(* Logix 5000 project; controller R1USB70001_CWRU_Scenario_Gen_20111116 vendor 1 type 14 code 54 rev 19.11; software revision 19.01; part 2 of 6 *)
(* tags used below, declared in another part *)
   ControlModePv : ControlModePv;
   DiscreteOutputsPv : DiscreteOutputsPv;
   ExecutePv : ExecutePv;
   Alternate_Control_Buffer : Output_Array;   // Array of bit-defined words from Alternate (external) Control source
   AP_GP_CH_SG1 : ALIAS FOR ACNR_GP_SG_N2:1:O.2;
   AP_GP_CH_SG2 : ALIAS FOR ACNR_GP_SG_N2:1:O.3;
   AP_GP_SR_SG1 : ALIAS FOR ACNR_GP_SG_N2:1:O.0;
   AP_GP_SR_SG2 : ALIAS FOR ACNR_GP_SG_N2:1:O.1;
   AS_SP_L1_SG1 : ALIAS FOR ACNR_SP_SG_N3:1:O.0;
   AS_SP_L1_SG2 : ALIAS FOR ACNR_SP_SG_N3:1:O.1;
   AS_SP_L2_SG1 : ALIAS FOR ACNR_SP_SG_N3:1:O.2;
   AS_SP_L2_SG2 : ALIAS FOR ACNR_SP_SG_N3:1:O.3;
   BuildTableIndex : DINT;
   CalcRemainTimeIndex : DINT;
   CalcTotalTimeIndex : DINT;
   CL_GP_SC_SG1 : ALIAS FOR ACNR_GP_SG_N2:5:O.0;
   CL_GP_SC_SG2 : ALIAS FOR ACNR_GP_SG_N2:5:O.1;
   CL_GP_SF_SG1 : ALIAS FOR ACNR_GP_SG_N2:5:O.2;
   CL_GP_SF_SG2 : ALIAS FOR ACNR_GP_SG_N2:5:O.3;
   CL_GP_WF_SG1 : ALIAS FOR ACNR_GP_SG_N2:5:O.6;
   CL_GP_WF_SG2 : ALIAS FOR ACNR_GP_SG_N2:5:O.7;
   CL_GP_WT_SG1 : ALIAS FOR ACNR_GP_SG_N2:5:O.4;
   CL_GP_WT_SG2 : ALIAS FOR ACNR_GP_SG_N2:5:O.5;
   ControlMode : ControlModePub;
   Execute : ExecutePub;
   HMI : HMIPub;
   IL_GP_SC_SG1 : ALIAS FOR ACNR_GP_SG_N2:6:O.0;
   IL_GP_SC_SG2 : ALIAS FOR ACNR_GP_SG_N2:6:O.1;
   IL_GP_SF_SG1 : ALIAS FOR ACNR_GP_SG_N2:6:O.2;
   IL_GP_SF_SG2 : ALIAS FOR ACNR_GP_SG_N2:6:O.3;
   IL_GP_WF_SG1 : ALIAS FOR ACNR_GP_SG_N2:6:O.6;
   IL_GP_WF_SG2 : ALIAS FOR ACNR_GP_SG_N2:6:O.7;
   IL_GP_WT_SG1 : ALIAS FOR ACNR_GP_SG_N2:6:O.4;
   IL_GP_WT_SG2 : ALIAS FOR ACNR_GP_SG_N2:6:O.5;
   RL_GP_SC_SG1 : ALIAS FOR ACNR_GP_SG_N2:4:O.0;
   RL_GP_SC_SG2 : ALIAS FOR ACNR_GP_SG_N2:4:O.1;
   RL_GP_SF_SG1 : ALIAS FOR ACNR_GP_SG_N2:4:O.2;
   RL_GP_SF_SG2 : ALIAS FOR ACNR_GP_SG_N2:4:O.3;
   RL_GP_WF_SG1 : ALIAS FOR ACNR_GP_SG_N2:4:O.6;
   RL_GP_WF_SG2 : ALIAS FOR ACNR_GP_SG_N2:4:O.7;
   RL_GP_WT_SG1 : ALIAS FOR ACNR_GP_SG_N2:4:O.4;
   RL_GP_WT_SG2 : ALIAS FOR ACNR_GP_SG_N2:4:O.5;
   RL_LP_B1_L1_SG1 : ALIAS FOR ACNR_RP_SG_N4:1:O.2;
   RL_LP_B1_L1_SG2 : ALIAS FOR ACNR_RP_SG_N4:1:O.3;
   RL_LP_B1_L2_SG1 : ALIAS FOR ACNR_RP_SG_N4:1:O.4;
   RL_LP_B1_L2_SG2 : ALIAS FOR ACNR_RP_SG_N4:1:O.5;
   RL_LP_B1_L3_SG1 : ALIAS FOR ACNR_RP_SG_N4:1:O.6;
   RL_LP_B1_L3_SG2 : ALIAS FOR ACNR_RP_SG_N4:1:O.7;
   RL_LP_B1_L4_SG1 : ALIAS FOR ACNR_RP_SG_N4:2:O.0;
   RL_LP_B1_L4_SG2 : ALIAS FOR ACNR_RP_SG_N4:2:O.1;
   RL_LP_B1_L5_SG1 : ALIAS FOR ACNR_RP_SG_N4:2:O.2;
   RL_LP_B1_SG : ALIAS FOR ACNR_RP_SG_N4:1:O.1;
   RL_LP_ML_SG : ALIAS FOR ACNR_RP_SG_N4:1:O.0;
   SC_GP_BT_SG1 : ALIAS FOR ACNR_GP_SG_N2:3:O.0;
   SC_GP_BT_SG2 : ALIAS FOR ACNR_GP_SG_N2:3:O.1;
   SC_GP_GD_SG1 : ALIAS FOR ACNR_GP_SG_N2:3:O.2;
   SC_GP_GD_SG2 : ALIAS FOR ACNR_GP_SG_N2:3:O.3;
   SC_SP_LN_SG1 : ALIAS FOR ACNR_SP_SG_N3:2:O.2;
   SC_SP_LN_SG2 : ALIAS FOR ACNR_SP_SG_N3:2:O.3;
   Scenario : Scenario_Def[100];
   SF_GP_BT_SG1 : ALIAS FOR ACNR_GP_SG_N2:2:O.4;
   SF_GP_BT_SG2 : ALIAS FOR ACNR_GP_SG_N2:2:O.5;
   SF_GP_GD_SG1 : ALIAS FOR ACNR_GP_SG_N2:2:O.6;
   SF_GP_GD_SG2 : ALIAS FOR ACNR_GP_SG_N2:2:O.7;
   SF_SP_LN_SG1 : ALIAS FOR ACNR_SP_SG_N3:2:O.0;
   SF_SP_LN_SG2 : ALIAS FOR ACNR_SP_SG_N3:2:O.1;
   TimeTblStepNmbr : DINT;
   WF_GP_BT_SG1 : ALIAS FOR ACNR_GP_SG_N2:1:O.4;
   WF_GP_BT_SG2 : ALIAS FOR ACNR_GP_SG_N2:1:O.5;
   WF_GP_GD_SG1 : ALIAS FOR ACNR_GP_SG_N2:1:O.6;
   WF_GP_GD_SG2 : ALIAS FOR ACNR_GP_SG_N2:1:O.7;
   WF_SP_LN_SG1 : ALIAS FOR ACNR_SP_SG_N3:1:O.4;
   WF_SP_LN_SG2 : ALIAS FOR ACNR_SP_SG_N3:1:O.5;
   WT_GP_BT_SG1 : ALIAS FOR ACNR_GP_SG_N2:2:O.0;
   WT_GP_BT_SG2 : ALIAS FOR ACNR_GP_SG_N2:2:O.1;
   WT_GP_GD_SG1 : ALIAS FOR ACNR_GP_SG_N2:2:O.2;
   WT_GP_GD_SG2 : ALIAS FOR ACNR_GP_SG_N2:2:O.3;
   WT_SP_LN_SG1 : ALIAS FOR ACNR_SP_SG_N3:1:O.6;
   WT_SP_LN_SG2 : ALIAS FOR ACNR_SP_SG_N3:1:O.7;
(* MainProgram, continued *)

ROUTINE BuildTimeTableStep   (* ladder *)
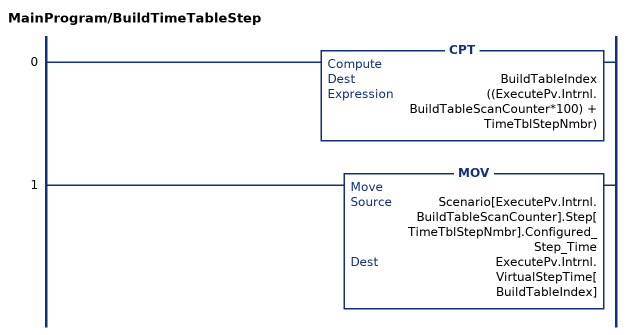
   0: CPT(BuildTableIndex,((ExecutePv.Intrnl.BuildTableScanCounter*100) + TimeTblStepNmbr));
   1: MOV(Scenario[ExecutePv.Intrnl.BuildTableScanCounter].Step[TimeTblStepNmbr].Configured_Step_Time,ExecutePv.Intrnl.VirtualStepTime[BuildTableIndex]);
END_ROUTINE

ROUTINE CalculateCampaignTime   (* ladder *)
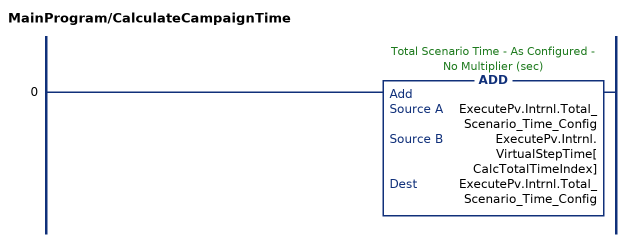
   0: ADD(ExecutePv.Intrnl.Total_Scenario_Time_Config,ExecutePv.Intrnl.VirtualStepTime[CalcTotalTimeIndex],ExecutePv.Intrnl.Total_Scenario_Time_Config);
END_ROUTINE

ROUTINE CalculateRemainingTime   (* ladder *)
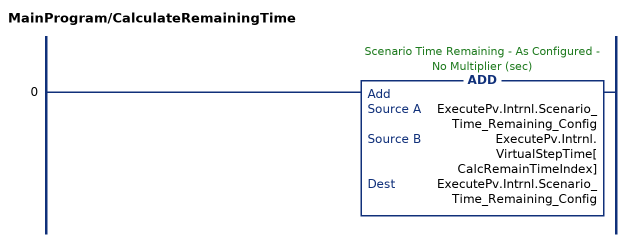
   0: ADD(ExecutePv.Intrnl.Scenario_Time_Remaining_Config,ExecutePv.Intrnl.VirtualStepTime[CalcRemainTimeIndex],ExecutePv.Intrnl.Scenario_Time_Remaining_Config);
END_ROUTINE

ROUTINE Control_Mode   (* ladder *)
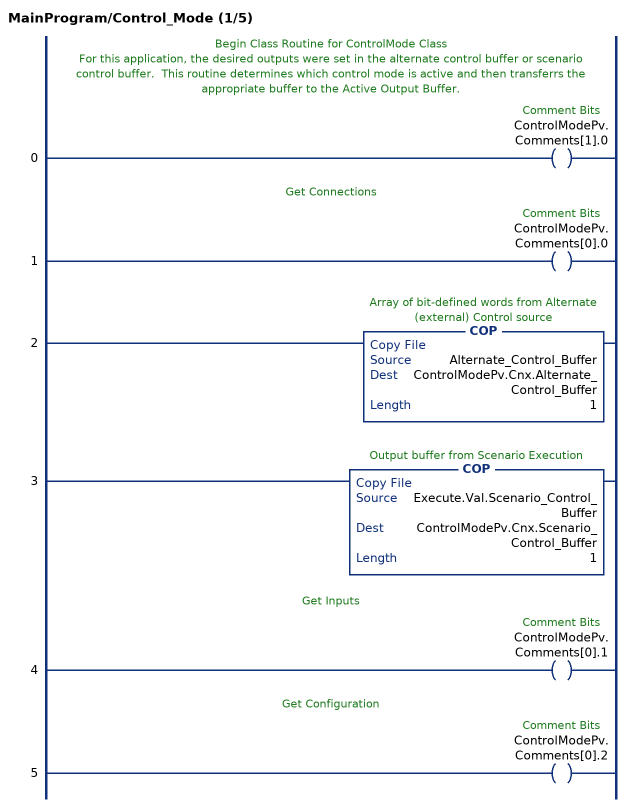
   // Begin Class Routine for ControlMode Class
   // For this application, the desired outputs were set in the alternate control buffer or scenario control buffer.  This routine determines which control mode is active and then transferrs the appropriate buffer to the Active Output Buffer.
   0: OTE(ControlModePv.Comments[1].0);
   // Get Connections
   1: OTE(ControlModePv.Comments[0].0);
   2: COP(Alternate_Control_Buffer,ControlModePv.Cnx.Alternate_Control_Buffer,1);
   3: COP(Execute.Val.Scenario_Control_Buffer,ControlModePv.Cnx.Scenario_Control_Buffer,1);
   // Get Inputs
   4: OTE(ControlModePv.Comments[0].1);
   // Get Configuration
   5: OTE(ControlModePv.Comments[0].2);
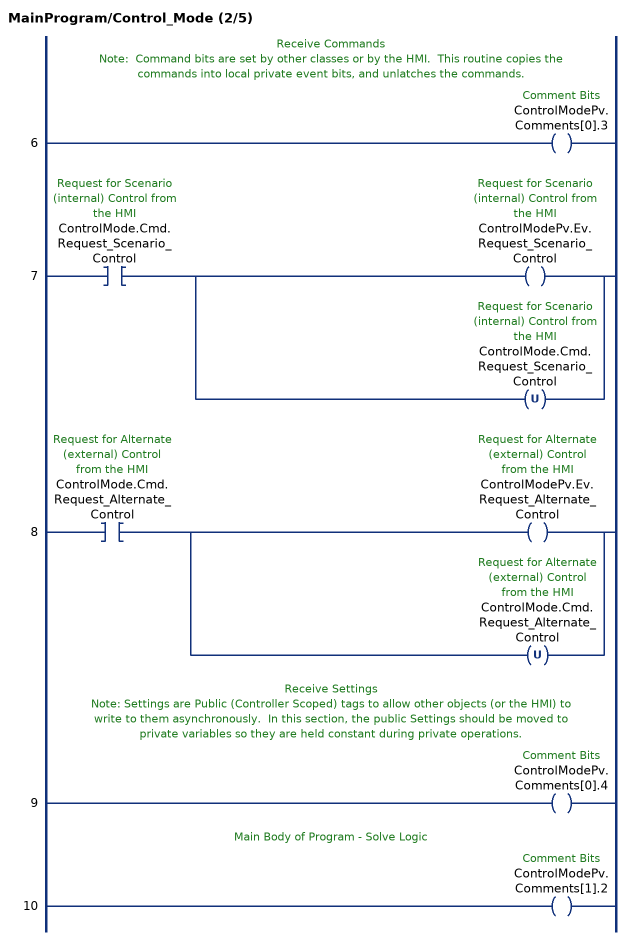
   // Receive Commands
   // Note:  Command bits are set by other classes or by the HMI.  This routine copies the commands into local private event bits, and unlatches the commands.
   6: OTE(ControlModePv.Comments[0].3);
   7: XIC(ControlMode.Cmd.Request_Scenario_Control)[OTE(ControlModePv.Ev.Request_Scenario_Control) ,OTU(ControlMode.Cmd.Request_Scenario_Control) ];
   8: XIC(ControlMode.Cmd.Request_Alternate_Control)[OTE(ControlModePv.Ev.Request_Alternate_Control) ,OTU(ControlMode.Cmd.Request_Alternate_Control) ];
   // Receive Settings
   // Note: Settings are Public (Controller Scoped) tags to allow other objects (or the HMI) to write to them asynchronously.  In this section, the public Settings should be moved to private variables so they are held constant during private operations.
   9: OTE(ControlModePv.Comments[0].4);
   // Main Body of Program - Solve Logic
   10: OTE(ControlModePv.Comments[1].2);
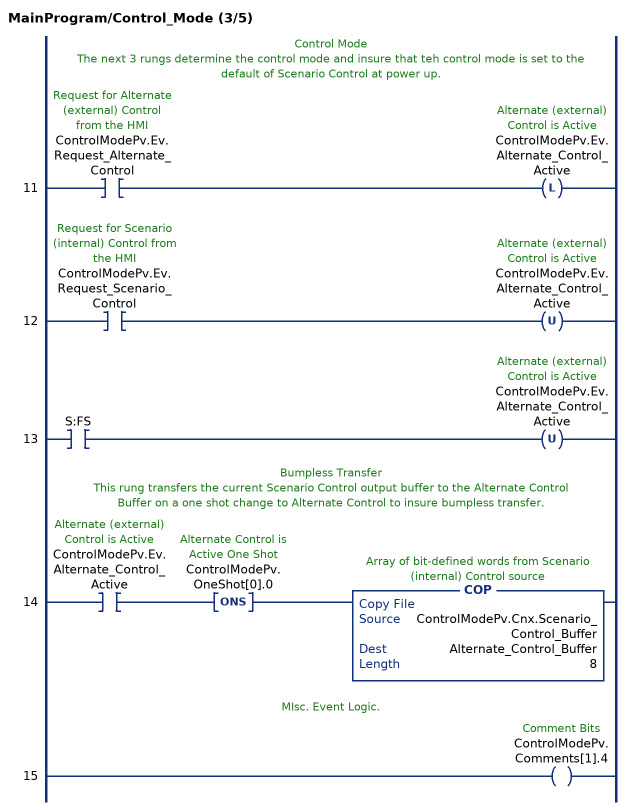
   // Control Mode
   // The next 3 rungs determine the control mode and insure that teh control mode is set to the default of Scenario Control at power up.
   11: XIC(ControlModePv.Ev.Request_Alternate_Control)OTL(ControlModePv.Ev.Alternate_Control_Active);
   12: XIC(ControlModePv.Ev.Request_Scenario_Control)OTU(ControlModePv.Ev.Alternate_Control_Active);
   13: XIC(S:FS)OTU(ControlModePv.Ev.Alternate_Control_Active);
   // Bumpless Transfer
   // This rung transfers the current Scenario Control output buffer to the Alternate Control Buffer on a one shot change to Alternate Control to insure bumpless transfer.
   14: XIC(ControlModePv.Ev.Alternate_Control_Active)ONS(ControlModePv.OneShot[0].0)COP(ControlModePv.Cnx.Scenario_Control_Buffer,Alternate_Control_Buffer,8);
   // MIsc. Event Logic.
   15: OTE(ControlModePv.Comments[1].4);
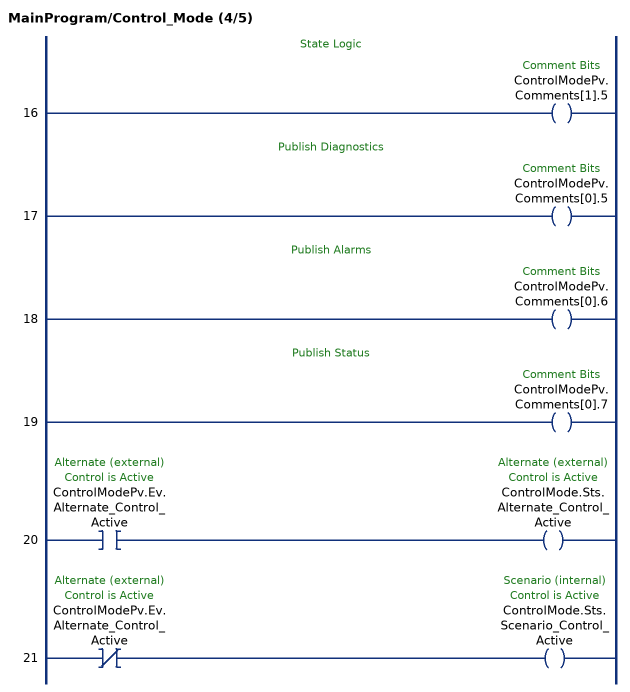
   // State Logic
   16: OTE(ControlModePv.Comments[1].5);
   // Publish Diagnostics
   17: OTE(ControlModePv.Comments[0].5);
   // Publish Alarms
   18: OTE(ControlModePv.Comments[0].6);
   // Publish Status
   19: OTE(ControlModePv.Comments[0].7);
   20: XIC(ControlModePv.Ev.Alternate_Control_Active)OTE(ControlMode.Sts.Alternate_Control_Active);
   21: XIO(ControlModePv.Ev.Alternate_Control_Active)OTE(ControlMode.Sts.Scenario_Control_Active);
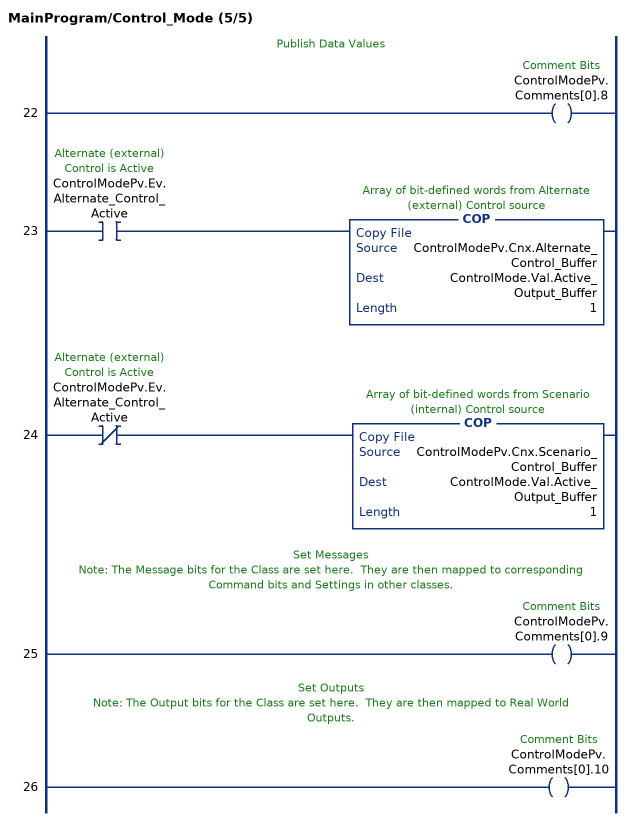
   // Publish Data Values
   22: OTE(ControlModePv.Comments[0].8);
   23: XIC(ControlModePv.Ev.Alternate_Control_Active)COP(ControlModePv.Cnx.Alternate_Control_Buffer,ControlMode.Val.Active_Output_Buffer,1);
   24: XIO(ControlModePv.Ev.Alternate_Control_Active)COP(ControlModePv.Cnx.Scenario_Control_Buffer,ControlMode.Val.Active_Output_Buffer,1);
   // Set Messages
   // Note: The Message bits for the Class are set here.  They are then mapped to corresponding Command bits and Settings in other classes.
   25: OTE(ControlModePv.Comments[0].9);
   // Set Outputs
   // Note: The Output bits for the Class are set here.  They are then mapped to Real World Outputs.
   26: OTE(ControlModePv.Comments[0].10);
END_ROUTINE

ROUTINE DiscreteOutputs   (* ladder *)
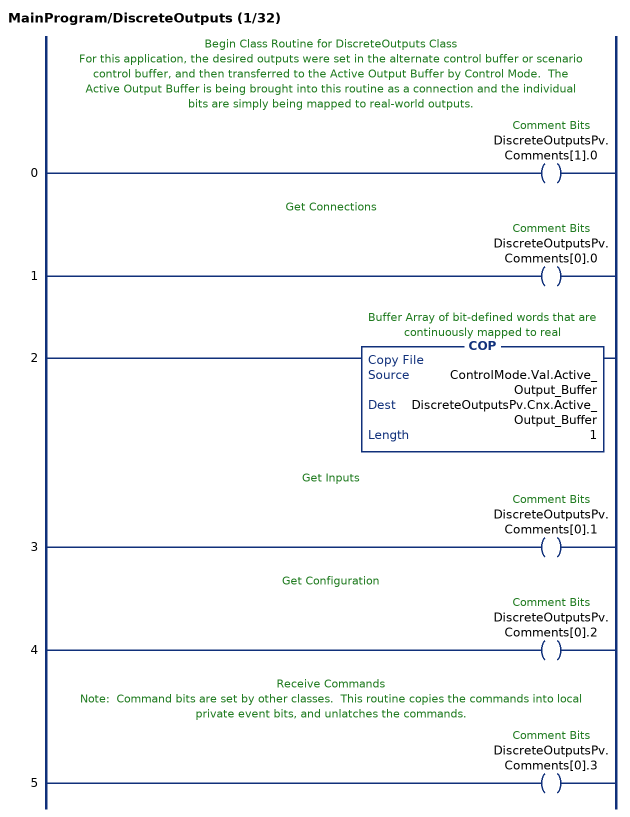
   // Begin Class Routine for DiscreteOutputs Class
   // For this application, the desired outputs were set in the alternate control buffer or scenario control buffer, and then transferred to the Active Output Buffer by Control Mode.  The Active Output Buffer is being brought into this routine as a connection and the individual bits are simply being mapped to real-world outputs.
   0: OTE(DiscreteOutputsPv.Comments[1].0);
   // Get Connections
   1: OTE(DiscreteOutputsPv.Comments[0].0);
   2: COP(ControlMode.Val.Active_Output_Buffer,DiscreteOutputsPv.Cnx.Active_Output_Buffer,1);
   // Get Inputs
   3: OTE(DiscreteOutputsPv.Comments[0].1);
   // Get Configuration
   4: OTE(DiscreteOutputsPv.Comments[0].2);
   // Receive Commands
   // Note:  Command bits are set by other classes.  This routine copies the commands into local private event bits, and unlatches the commands.
   5: OTE(DiscreteOutputsPv.Comments[0].3);
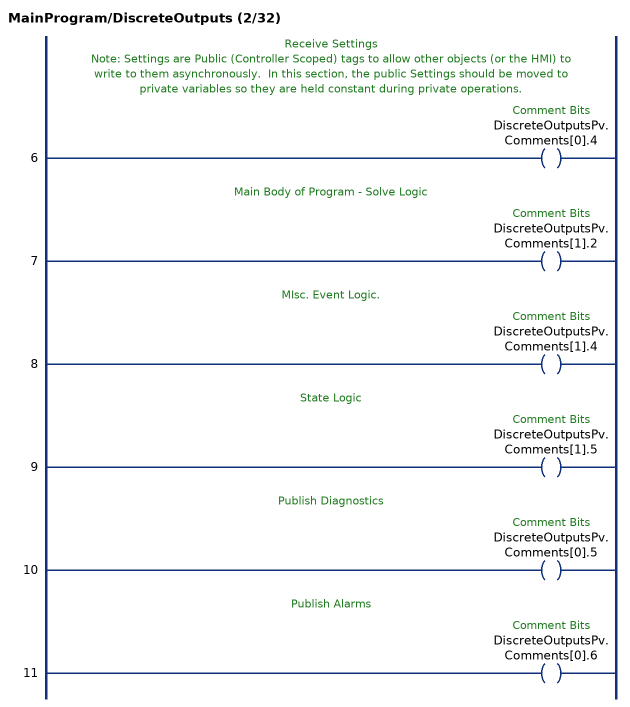
   // Receive Settings
   // Note: Settings are Public (Controller Scoped) tags to allow other objects (or the HMI) to write to them asynchronously.  In this section, the public Settings should be moved to private variables so they are held constant during private operations.
   6: OTE(DiscreteOutputsPv.Comments[0].4);
   // Main Body of Program - Solve Logic
   7: OTE(DiscreteOutputsPv.Comments[1].2);
   // MIsc. Event Logic.
   8: OTE(DiscreteOutputsPv.Comments[1].4);
   // State Logic
   9: OTE(DiscreteOutputsPv.Comments[1].5);
   // Publish Diagnostics
   10: OTE(DiscreteOutputsPv.Comments[0].5);
   // Publish Alarms
   11: OTE(DiscreteOutputsPv.Comments[0].6);
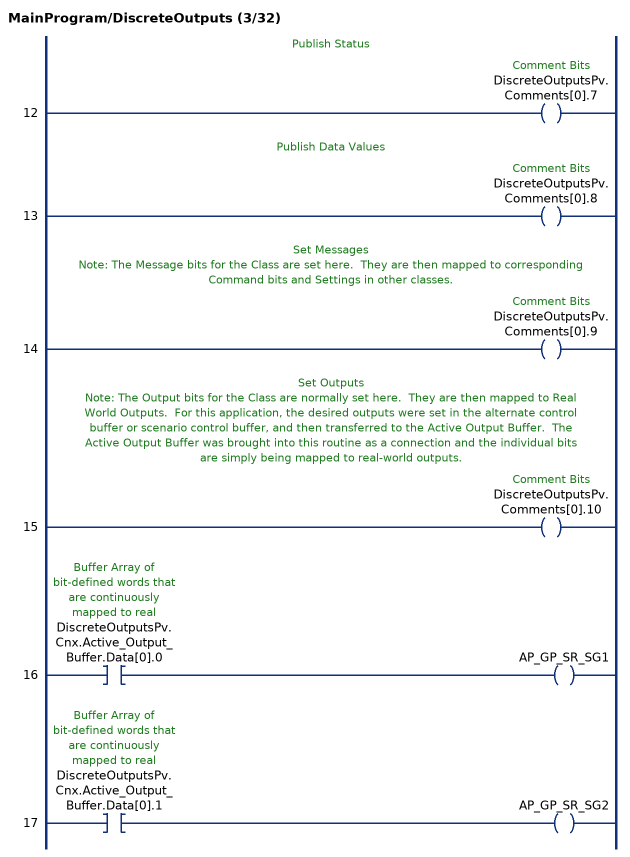
   // Publish Status
   12: OTE(DiscreteOutputsPv.Comments[0].7);
   // Publish Data Values
   13: OTE(DiscreteOutputsPv.Comments[0].8);
   // Set Messages
   // Note: The Message bits for the Class are set here.  They are then mapped to corresponding Command bits and Settings in other classes.
   14: OTE(DiscreteOutputsPv.Comments[0].9);
   // Set Outputs
   // Note: The Output bits for the Class are normally set here.  They are then mapped to Real World Outputs.  For this application, the desired outputs were set in the alternate control buffer or scenario control buffer, and then transferred to the Active Output Buffer.  The Active Output Buffer was brought into this routine as a connection and the individual bits are simply being mapped to real-world outputs.
   15: OTE(DiscreteOutputsPv.Comments[0].10);
   16: XIC(DiscreteOutputsPv.Cnx.Active_Output_Buffer.Data[0].0)OTE(AP_GP_SR_SG1);
   17: XIC(DiscreteOutputsPv.Cnx.Active_Output_Buffer.Data[0].1)OTE(AP_GP_SR_SG2);
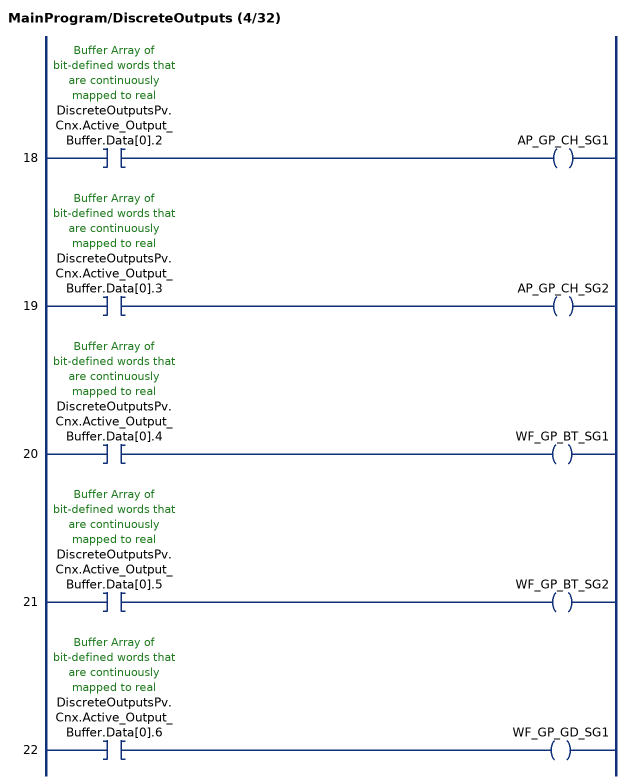
   18: XIC(DiscreteOutputsPv.Cnx.Active_Output_Buffer.Data[0].2)OTE(AP_GP_CH_SG1);
   19: XIC(DiscreteOutputsPv.Cnx.Active_Output_Buffer.Data[0].3)OTE(AP_GP_CH_SG2);
   20: XIC(DiscreteOutputsPv.Cnx.Active_Output_Buffer.Data[0].4)OTE(WF_GP_BT_SG1);
   21: XIC(DiscreteOutputsPv.Cnx.Active_Output_Buffer.Data[0].5)OTE(WF_GP_BT_SG2);
   22: XIC(DiscreteOutputsPv.Cnx.Active_Output_Buffer.Data[0].6)OTE(WF_GP_GD_SG1);
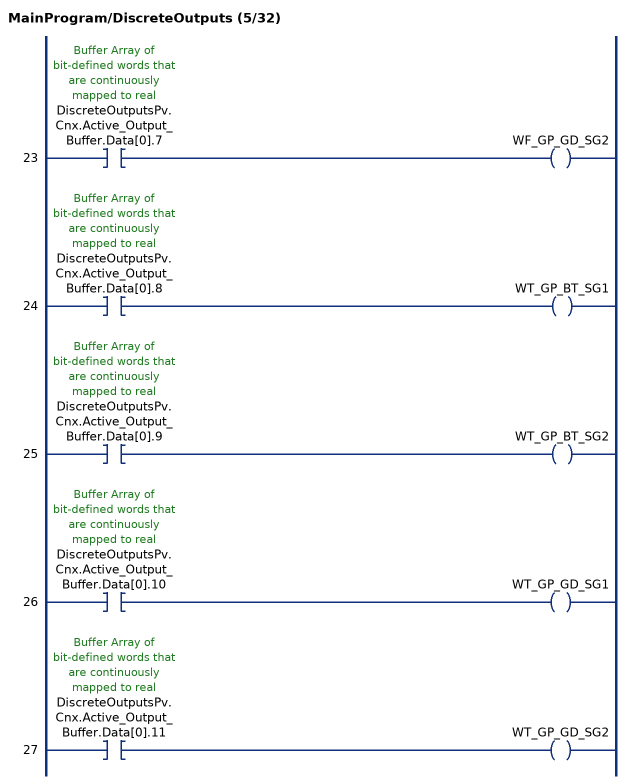
   23: XIC(DiscreteOutputsPv.Cnx.Active_Output_Buffer.Data[0].7)OTE(WF_GP_GD_SG2);
   24: XIC(DiscreteOutputsPv.Cnx.Active_Output_Buffer.Data[0].8)OTE(WT_GP_BT_SG1);
   25: XIC(DiscreteOutputsPv.Cnx.Active_Output_Buffer.Data[0].9)OTE(WT_GP_BT_SG2);
   26: XIC(DiscreteOutputsPv.Cnx.Active_Output_Buffer.Data[0].10)OTE(WT_GP_GD_SG1);
   27: XIC(DiscreteOutputsPv.Cnx.Active_Output_Buffer.Data[0].11)OTE(WT_GP_GD_SG2);
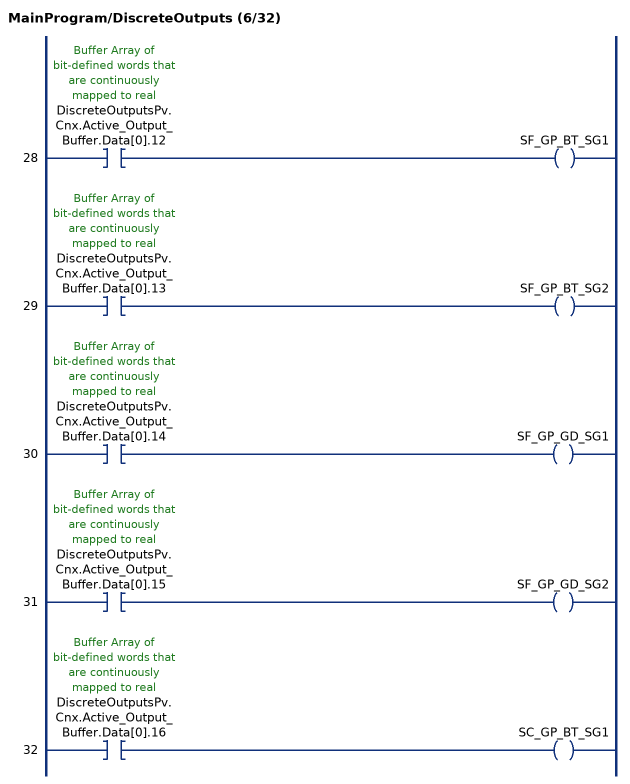
   28: XIC(DiscreteOutputsPv.Cnx.Active_Output_Buffer.Data[0].12)OTE(SF_GP_BT_SG1);
   29: XIC(DiscreteOutputsPv.Cnx.Active_Output_Buffer.Data[0].13)OTE(SF_GP_BT_SG2);
   30: XIC(DiscreteOutputsPv.Cnx.Active_Output_Buffer.Data[0].14)OTE(SF_GP_GD_SG1);
   31: XIC(DiscreteOutputsPv.Cnx.Active_Output_Buffer.Data[0].15)OTE(SF_GP_GD_SG2);
   32: XIC(DiscreteOutputsPv.Cnx.Active_Output_Buffer.Data[0].16)OTE(SC_GP_BT_SG1);
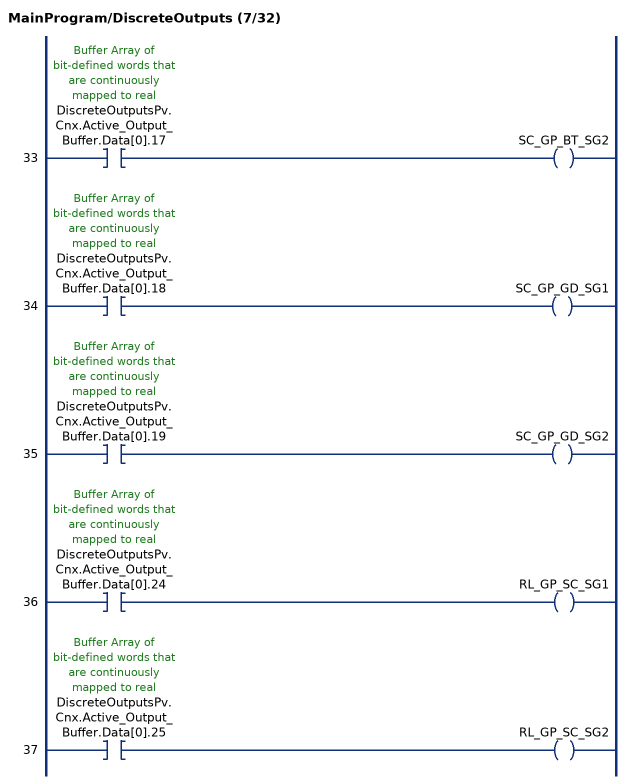
   33: XIC(DiscreteOutputsPv.Cnx.Active_Output_Buffer.Data[0].17)OTE(SC_GP_BT_SG2);
   34: XIC(DiscreteOutputsPv.Cnx.Active_Output_Buffer.Data[0].18)OTE(SC_GP_GD_SG1);
   35: XIC(DiscreteOutputsPv.Cnx.Active_Output_Buffer.Data[0].19)OTE(SC_GP_GD_SG2);
   36: XIC(DiscreteOutputsPv.Cnx.Active_Output_Buffer.Data[0].24)OTE(RL_GP_SC_SG1);
   37: XIC(DiscreteOutputsPv.Cnx.Active_Output_Buffer.Data[0].25)OTE(RL_GP_SC_SG2);
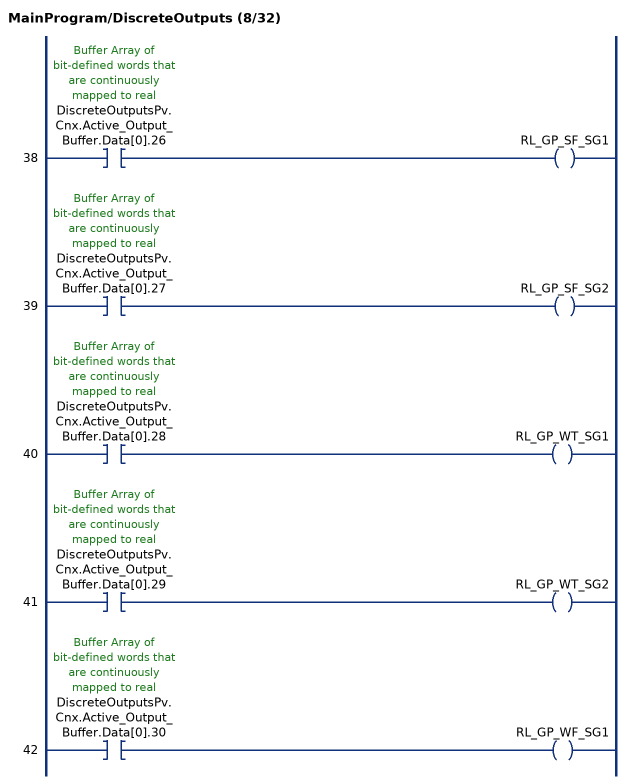
   38: XIC(DiscreteOutputsPv.Cnx.Active_Output_Buffer.Data[0].26)OTE(RL_GP_SF_SG1);
   39: XIC(DiscreteOutputsPv.Cnx.Active_Output_Buffer.Data[0].27)OTE(RL_GP_SF_SG2);
   40: XIC(DiscreteOutputsPv.Cnx.Active_Output_Buffer.Data[0].28)OTE(RL_GP_WT_SG1);
   41: XIC(DiscreteOutputsPv.Cnx.Active_Output_Buffer.Data[0].29)OTE(RL_GP_WT_SG2);
   42: XIC(DiscreteOutputsPv.Cnx.Active_Output_Buffer.Data[0].30)OTE(RL_GP_WF_SG1);
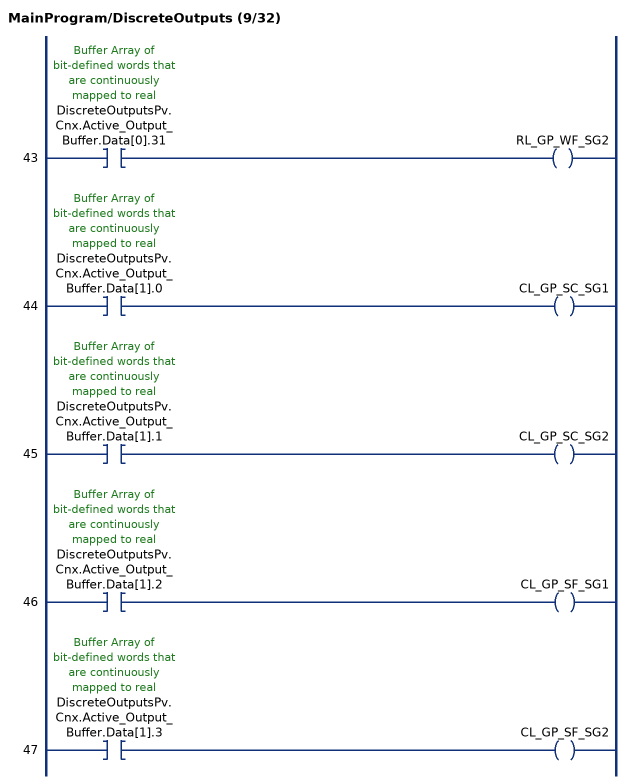
   43: XIC(DiscreteOutputsPv.Cnx.Active_Output_Buffer.Data[0].31)OTE(RL_GP_WF_SG2);
   44: XIC(DiscreteOutputsPv.Cnx.Active_Output_Buffer.Data[1].0)OTE(CL_GP_SC_SG1);
   45: XIC(DiscreteOutputsPv.Cnx.Active_Output_Buffer.Data[1].1)OTE(CL_GP_SC_SG2);
   46: XIC(DiscreteOutputsPv.Cnx.Active_Output_Buffer.Data[1].2)OTE(CL_GP_SF_SG1);
   47: XIC(DiscreteOutputsPv.Cnx.Active_Output_Buffer.Data[1].3)OTE(CL_GP_SF_SG2);
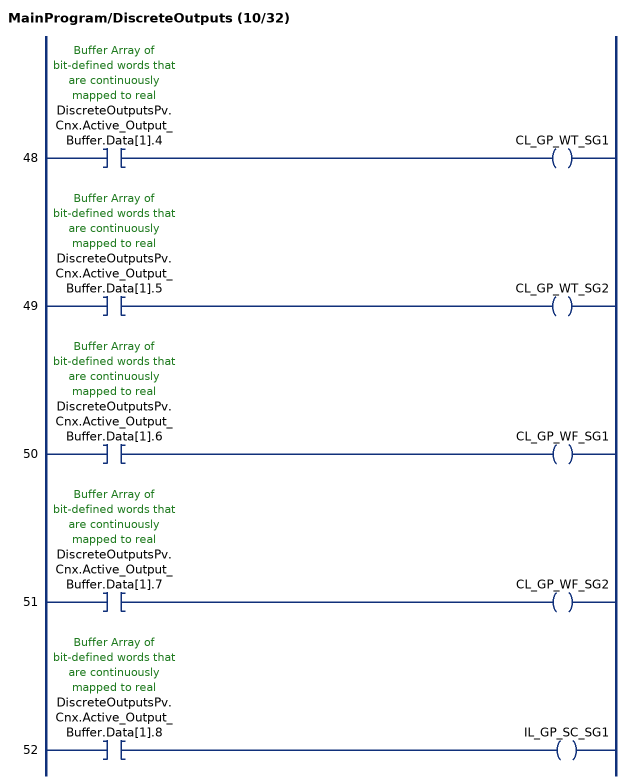
   48: XIC(DiscreteOutputsPv.Cnx.Active_Output_Buffer.Data[1].4)OTE(CL_GP_WT_SG1);
   49: XIC(DiscreteOutputsPv.Cnx.Active_Output_Buffer.Data[1].5)OTE(CL_GP_WT_SG2);
   50: XIC(DiscreteOutputsPv.Cnx.Active_Output_Buffer.Data[1].6)OTE(CL_GP_WF_SG1);
   51: XIC(DiscreteOutputsPv.Cnx.Active_Output_Buffer.Data[1].7)OTE(CL_GP_WF_SG2);
   52: XIC(DiscreteOutputsPv.Cnx.Active_Output_Buffer.Data[1].8)OTE(IL_GP_SC_SG1);
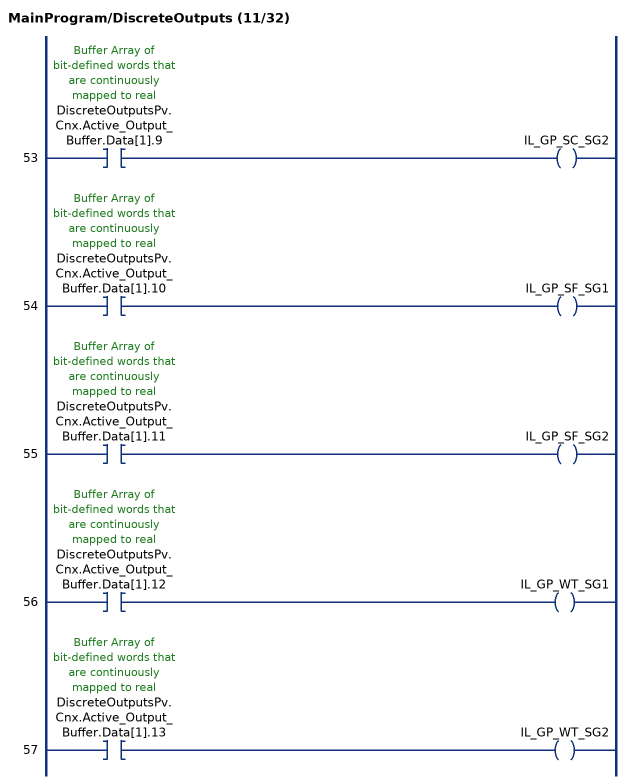
   53: XIC(DiscreteOutputsPv.Cnx.Active_Output_Buffer.Data[1].9)OTE(IL_GP_SC_SG2);
   54: XIC(DiscreteOutputsPv.Cnx.Active_Output_Buffer.Data[1].10)OTE(IL_GP_SF_SG1);
   55: XIC(DiscreteOutputsPv.Cnx.Active_Output_Buffer.Data[1].11)OTE(IL_GP_SF_SG2);
   56: XIC(DiscreteOutputsPv.Cnx.Active_Output_Buffer.Data[1].12)OTE(IL_GP_WT_SG1);
   57: XIC(DiscreteOutputsPv.Cnx.Active_Output_Buffer.Data[1].13)OTE(IL_GP_WT_SG2);
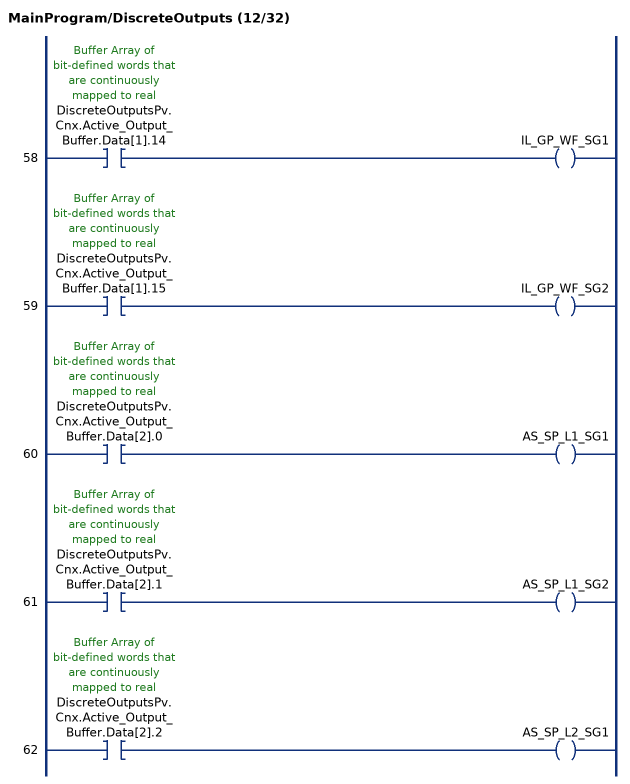
   58: XIC(DiscreteOutputsPv.Cnx.Active_Output_Buffer.Data[1].14)OTE(IL_GP_WF_SG1);
   59: XIC(DiscreteOutputsPv.Cnx.Active_Output_Buffer.Data[1].15)OTE(IL_GP_WF_SG2);
   60: XIC(DiscreteOutputsPv.Cnx.Active_Output_Buffer.Data[2].0)OTE(AS_SP_L1_SG1);
   61: XIC(DiscreteOutputsPv.Cnx.Active_Output_Buffer.Data[2].1)OTE(AS_SP_L1_SG2);
   62: XIC(DiscreteOutputsPv.Cnx.Active_Output_Buffer.Data[2].2)OTE(AS_SP_L2_SG1);
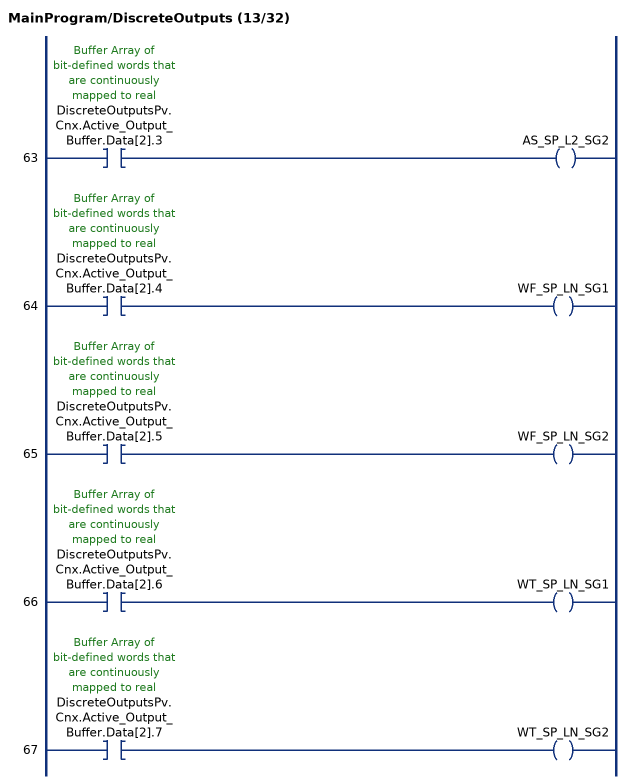
   63: XIC(DiscreteOutputsPv.Cnx.Active_Output_Buffer.Data[2].3)OTE(AS_SP_L2_SG2);
   64: XIC(DiscreteOutputsPv.Cnx.Active_Output_Buffer.Data[2].4)OTE(WF_SP_LN_SG1);
   65: XIC(DiscreteOutputsPv.Cnx.Active_Output_Buffer.Data[2].5)OTE(WF_SP_LN_SG2);
   66: XIC(DiscreteOutputsPv.Cnx.Active_Output_Buffer.Data[2].6)OTE(WT_SP_LN_SG1);
   67: XIC(DiscreteOutputsPv.Cnx.Active_Output_Buffer.Data[2].7)OTE(WT_SP_LN_SG2);
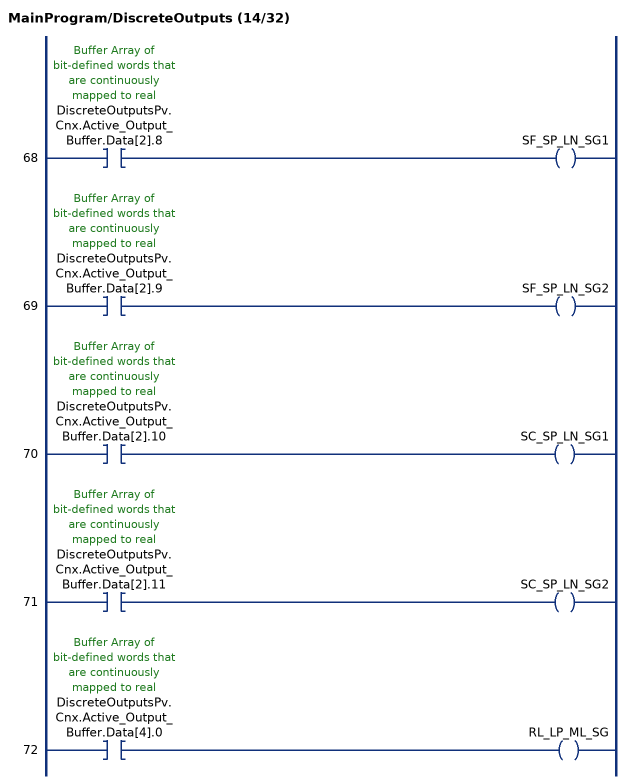
   68: XIC(DiscreteOutputsPv.Cnx.Active_Output_Buffer.Data[2].8)OTE(SF_SP_LN_SG1);
   69: XIC(DiscreteOutputsPv.Cnx.Active_Output_Buffer.Data[2].9)OTE(SF_SP_LN_SG2);
   70: XIC(DiscreteOutputsPv.Cnx.Active_Output_Buffer.Data[2].10)OTE(SC_SP_LN_SG1);
   71: XIC(DiscreteOutputsPv.Cnx.Active_Output_Buffer.Data[2].11)OTE(SC_SP_LN_SG2);
   72: XIC(DiscreteOutputsPv.Cnx.Active_Output_Buffer.Data[4].0)OTE(RL_LP_ML_SG);
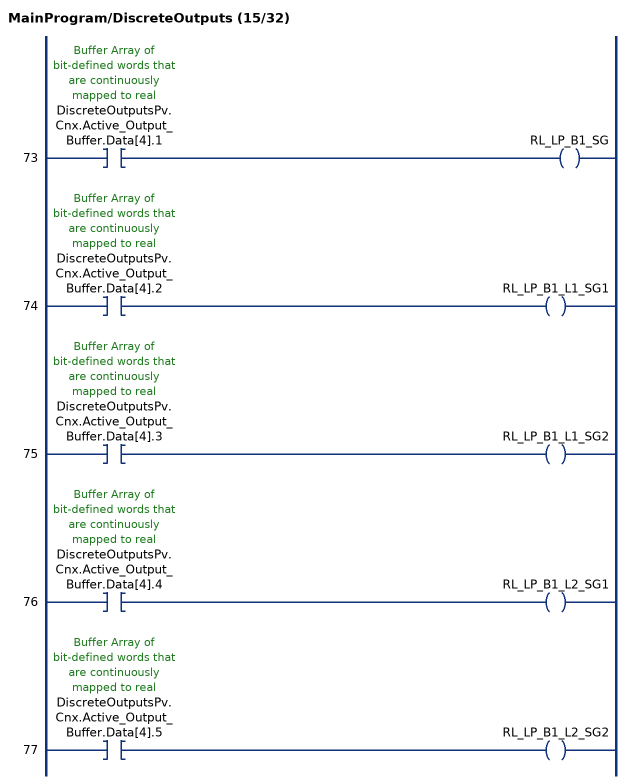
   73: XIC(DiscreteOutputsPv.Cnx.Active_Output_Buffer.Data[4].1)OTE(RL_LP_B1_SG);
   74: XIC(DiscreteOutputsPv.Cnx.Active_Output_Buffer.Data[4].2)OTE(RL_LP_B1_L1_SG1);
   75: XIC(DiscreteOutputsPv.Cnx.Active_Output_Buffer.Data[4].3)OTE(RL_LP_B1_L1_SG2);
   76: XIC(DiscreteOutputsPv.Cnx.Active_Output_Buffer.Data[4].4)OTE(RL_LP_B1_L2_SG1);
   77: XIC(DiscreteOutputsPv.Cnx.Active_Output_Buffer.Data[4].5)OTE(RL_LP_B1_L2_SG2);
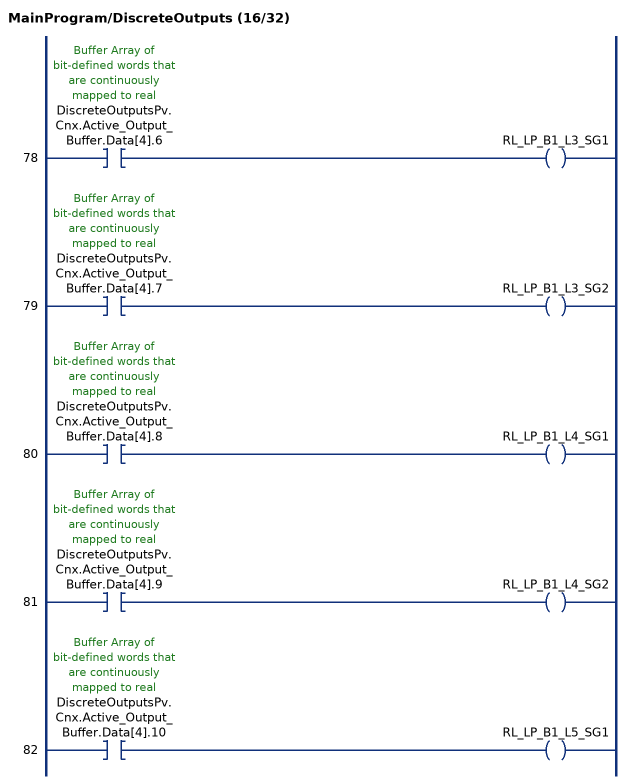
   78: XIC(DiscreteOutputsPv.Cnx.Active_Output_Buffer.Data[4].6)OTE(RL_LP_B1_L3_SG1);
   79: XIC(DiscreteOutputsPv.Cnx.Active_Output_Buffer.Data[4].7)OTE(RL_LP_B1_L3_SG2);
   80: XIC(DiscreteOutputsPv.Cnx.Active_Output_Buffer.Data[4].8)OTE(RL_LP_B1_L4_SG1);
   81: XIC(DiscreteOutputsPv.Cnx.Active_Output_Buffer.Data[4].9)OTE(RL_LP_B1_L4_SG2);
   82: XIC(DiscreteOutputsPv.Cnx.Active_Output_Buffer.Data[4].10)OTE(RL_LP_B1_L5_SG1);
